// TwinCAT 3 PLC project controller
// ProgramVersion: 3.1.4024.0
// libraries:
//   mobject-collections, * (mobject)
//   mobject-commands, * (mobject)
//   mobject-disposable, * (mobject)
//   mobject-enumerable, * (mobject)
//   Tc2_ModbusSrv, * (Beckhoff Automation GmbH)
//   Tc3_Module, * (Beckhoff Automation GmbH)
//   Tc3_System, * (Beckhoff Automation GmbH)
// project tree:
//   Lib/ModbusTwin/ BasicModbusDigitalTwin.TcPOU
//   Lib/Modbus/ ModbusCommand.TcPOU, ReadRegistersCommand.TcPOU, WriteSingleRegisterCommand.TcPOU
//   Programs/ Main.TcPOU
//   Programs/TestTwin/ TestTwin.TcPOU, TestSlaveConfigData.TcDUT, TestSlaveFastDataA.TcDUT, TestSlaveFastDataB.TcDUT
//   _Tasks/ PlcTask.TcTTO (not stored)
// real-time tasks:
//   TASK PlcTask: cycle T#10ms, priority 20, ADS port 350

// ---- Programs/TestTwin/TestSlaveConfigData.TcDUT
TYPE TestSlaveConfigData :
STRUCT
	config1 : INT;
	config2 : INT;
END_STRUCT
END_TYPE

// ---- Programs/TestTwin/TestSlaveFastDataA.TcDUT
TYPE TestSlaveFastDataA :
STRUCT
	fastData1 : INT;
	fastData2 : INT;
END_STRUCT
END_TYPE

// ---- Programs/TestTwin/TestSlaveFastDataB.TcDUT
TYPE TestSlaveFastDataB :
STRUCT
	fastData3 : INT;
	fastData4 : INT;
END_STRUCT
END_TYPE

// ---- Lib/ModbusTwin/BasicModbusDigitalTwin.TcPOU
{attribute 'linkalways'} 
{attribute 'no_explicit_call' := 'This FB is a CLASS and must be accessed using methods or properties'}
{attribute 'enable_dynamic_creation'}
FUNCTION_BLOCK ABSTRACT BasicModbusDigitalTwin
VAR
	ipAddress : STRING(15);
	tcpPort : UINT := MODBUS_TCP_PORT;
	unitId : USINT;	

	cyclicCommands : LinkedList;
	queuedCommands : Queue;
	
	commandRunner : SingleAsyncCommandRunner;
	currentCommand : I_AsyncCommand;
END_VAR

METHOD PRIVATE AddCyclicalCommand
VAR_INPUT
	command : I_AsyncCommand;
END_VAR
cyclicCommands.AddItem(command);
END_METHOD

METHOD PROTECTED AddCyclicalReadRegisters
VAR_INPUT
	modbusAddress : UINT;
	quantity : UINT (1..128);	
	destinationAddress : POINTER TO BYTE;
	destinationLength : UDINT;
	timeout : TIME;
END_VAR
VAR
	_modbusAddress : UINT;
	_quantity : UINT (1..128);	
	_destinationAddress : POINTER TO BYTE;
	_destinationLength : UDINT;
	_timeout : TIME;
	pCommand : POINTER TO ReadRegistersCommand;
	command : I_AsyncCommand;
END_VAR
_modbusAddress := modbusAddress;
_quantity := quantity;
_destinationAddress := destinationAddress;
_destinationLength := destinationLength;
_timeout := timeout;

pCommand := __NEW(ReadRegistersCommand(
	ipAddress := THIS^.ipAddress, tcpPort := THIS^.tcpPort, unitId := THIS^.unitId,
	modbusAddress := _modbusAddress, quantity := _quantity,
	destinationAddress := _destinationAddress, destinationLength := _destinationLength,
	timeout := _timeout));
command := pCommand^;
AddCyclicalCommand(command);
END_METHOD

METHOD PUBLIC CyclicCall
VAR_INST
	cyclicEnumerator : I_ForwardEnumerator;

END_VAR
IF cyclicEnumerator = 0 THEN
	cyclicEnumerator := cyclicCommands.GetEnumerator();
END_IF

IF NOT commandRunner.Busy THEN
	IF queuedCommands.Count > 0 THEN
		IF queuedCommands.TryDequeue(currentCommand) THEN
			commandRunner.ExecuteCommand(currentCommand);
		END_IF		
	ELSE
		IF cyclicEnumerator.MoveNext() AND_THEN cyclicEnumerator.TryGet(currentCommand) THEN
			commandRunner.ExecuteCommand(currentCommand);
		ELSE
			cyclicEnumerator.Dispose();
			cyclicEnumerator := 0;
		END_IF
	END_IF
END_IF

commandRunner.CyclicCall();
END_METHOD

METHOD FB_init : BOOL
VAR_INPUT
	bInitRetains : BOOL; // if TRUE, the retain variables are initialized (warm start / cold start)
	bInCopyCode : BOOL;  // if TRUE, the instance afterwards gets moved into the copy code (online change)
	ipAddress : STRING(15);
	tcpPort : UINT := MODBUS_TCP_PORT;
	unitId : USINT;
END_VAR
THIS^.ipAddress := ipAddress;
THIS^.tcpPort := tcpPort;
THIS^.unitId := unitId;
END_METHOD

METHOD PRIVATE QueueCommand
VAR_INPUT
	command : I_AsyncCommand;
END_VAR
queuedCommands.Enqueue(command);
END_METHOD

METHOD PROTECTED QueueWriteSingleCoil
VAR_INPUT
	modbusAddress : WORD;
	value : BOOL;
	timeout : TIME;
END_VAR
VAR
	pCommand : POINTER TO WriteSingleRegisterCommand;
	command : I_AsyncCommand;
END_VAR
END_METHOD

METHOD PROTECTED QueueWriteSingleRegister
VAR_INPUT
	modbusAddress : UINT;
	data : WORD;
	timeout : TIME;
END_VAR
VAR
	_modbusAddress : UINT;
	_data : WORD;
	_timeout : TIME;
	pCommand : POINTER TO WriteSingleRegisterCommand;
	command : I_AsyncCommand;
END_VAR
_modbusAddress := modbusAddress;
_data := data;
_timeout := timeout;

pCommand := __NEW(WriteSingleRegisterCommand(
	ipAddress := THIS^.ipAddress, tcpPort := THIS^.tcpPort, unitId := THIS^.unitId,
	modbusAddress := _modbusAddress, data := _data,
	timeout := _timeout));
command := pCommand^;
QueueCommand(command);
END_METHOD

END_FUNCTION_BLOCK

// ---- Lib/Modbus/ReadRegistersCommand.TcPOU
{attribute 'linkalways'} 
{attribute 'no_explicit_call' := 'This FB is a CLASS and must be accessed using methods or properties'}
{attribute 'enable_dynamic_creation'}
FUNCTION_BLOCK ReadRegistersCommand EXTENDS ModbusCommand
VAR
	fb : FB_MBReadRegs;
END_VAR

METHOD FB_init : BOOL
VAR_INPUT
	bInitRetains : BOOL; // if TRUE, the retain variables are initialized (warm start / cold start)
	bInCopyCode : BOOL;  // if TRUE, the instance afterwards gets moved into the copy code (online change)
	ipAddress : STRING(15);
	tcpPort : UINT := MODBUS_TCP_PORT;
	unitId : USINT;
	modbusAddress : UINT;
	quantity : UINT (1..128);
	destinationAddress : POINTER TO BYTE;
	destinationLength : UDINT;
	timeout : TIME;
END_VAR
fb.sIPAddr := ipAddress;
fb.nTCPPort := tcpPort;
fb.nUnitID := USINT_TO_BYTE(unitId);
fb.nMBAddr := UINT_TO_WORD(modbusAddress);
fb.nQuantity := UINT_TO_WORD(quantity);
fb.pDestAddr := destinationAddress;
fb.cbLength := destinationLength;
fb.tTimeout := timeout;
END_METHOD

METHOD PROTECTED OnAborting
VAR_INPUT
	StateControl : I_AsyncCommandStateControl;
END_VAR
fb(bExecute := FALSE);
StateControl.Next();
END_METHOD

METHOD PROTECTED OnCompleting
VAR_INPUT
	StateControl : I_AsyncCommandStateControl;
END_VAR
fb(bExecute := FALSE);
StateControl.Next();
END_METHOD

METHOD PROTECTED OnErrored
fb(bExecute := FALSE);
END_METHOD

METHOD PROTECTED OnExecuting
VAR_INPUT
	StateControl : I_AsyncCommandStateControl;
END_VAR
fb(bExecute := TRUE);

IF NOT fb.bBusy THEN
	IF fb.bError THEN
		StateControl.Error(fb.nErrId);
	ELSE
		StateControl.Next();
	END_IF
END_IF
END_METHOD

METHOD PROTECTED OnIdle
fb(bExecute := FALSE);
END_METHOD

METHOD PROTECTED OnInitializing
VAR_INPUT
	StateControl : I_AsyncCommandStateControl;
END_VAR
fb(bExecute := TRUE);
StateControl.Next();
END_METHOD

END_FUNCTION_BLOCK

// ---- Lib/Modbus/ModbusCommand.TcPOU
{attribute 'linkalways'} 
{attribute 'no_explicit_call' := 'This FB is a CLASS and must be accessed using methods or properties'}
{attribute 'enable_dynamic_creation'}
FUNCTION_BLOCK ABSTRACT ModbusCommand EXTENDS AsyncCommand IMPLEMENTS I_Disposable

METHOD Dispose
__DELETE(THIS);
END_METHOD

METHOD FB_exit : BOOL
VAR_INPUT
	bInCopyCode : BOOL; // if TRUE, the exit method is called for exiting an instance that is copied afterwards (online change).
END_VAR
// by default you would return if this is an in copy code, i.e. online change to this class
IF bInCopyCode THEN
	RETURN;
END_IF

// A word of warning. FB_exit does not NOT operate in the same way as a typical inherited method. If a child class does not implement FB_exit then it does not
// gain this one for itself. 
// The system will automatically call each FB_exit on each layer of inheritance one by one, starting with the child class and making it's way to the parent.
// Therefore code in here will only be triggered once the system reaches this layer of the object's deletion. The child class and all of it's variables
// will already have had FB_exit called by the time we reach this point!
END_METHOD

END_FUNCTION_BLOCK

// ---- Lib/Modbus/WriteSingleRegisterCommand.TcPOU
{attribute 'linkalways'} 
{attribute 'no_explicit_call' := 'This FB is a CLASS and must be accessed using methods or properties'}
{attribute 'enable_dynamic_creation'}
FUNCTION_BLOCK WriteSingleRegisterCommand EXTENDS ModbusCommand
VAR
	fb : FB_MBWriteSingleReg;
END_VAR

METHOD FB_init : BOOL
VAR_INPUT
	bInitRetains : BOOL; // if TRUE, the retain variables are initialized (warm start / cold start)
	bInCopyCode : BOOL;  // if TRUE, the instance afterwards gets moved into the copy code (online change)
	ipAddress : STRING(15);
	tcpPort : UINT := MODBUS_TCP_PORT;
	unitId : USINT;
	modbusAddress : UINT;
	data : WORD;
	timeout : TIME;
END_VAR
fb.sIPAddr := ipAddress;
fb.nTCPPort := tcpPort;
fb.nUnitID := USINT_TO_BYTE(unitId);
fb.nMBAddr := UINT_TO_WORD(modbusAddress);
fb.nValue := data;
fb.tTimeout := timeout;
END_METHOD

METHOD PROTECTED OnAborting
VAR_INPUT
	StateControl : I_AsyncCommandStateControl;
END_VAR
fb(bExecute := FALSE);
StateControl.Next();
END_METHOD

METHOD PROTECTED OnCompleting
VAR_INPUT
	StateControl : I_AsyncCommandStateControl;
END_VAR
fb(bExecute := FALSE);
StateControl.Next();
END_METHOD

METHOD PROTECTED OnExecuting
VAR_INPUT
	StateControl : I_AsyncCommandStateControl;
END_VAR
fb(bExecute := TRUE);

IF NOT fb.bBusy THEN
	IF fb.bError THEN
		StateControl.Error(fb.nErrId);
	ELSE
		StateControl.Next();
	END_IF
END_IF
END_METHOD

METHOD PROTECTED OnIdle
fb(bExecute := FALSE);
END_METHOD

METHOD PROTECTED OnInitializing
VAR_INPUT
	StateControl : I_AsyncCommandStateControl;
END_VAR
fb(bExecute := TRUE);
StateControl.Next();
END_METHOD

END_FUNCTION_BLOCK

// ---- Programs/Main.TcPOU
PROGRAM Main
VAR
	testSlave : TestTwin(ipAddress := '127.0.0.1', tcpPort := 503, unitId := 255);
END_VAR

testSlave.CyclicCall();

END_PROGRAM

// ---- Programs/TestTwin/TestTwin.TcPOU
{attribute 'linkalways'} 
{attribute 'no_explicit_call' := 'This FB is a CLASS and must be accessed using methods or properties'}
{attribute 'enable_dynamic_creation'}
FUNCTION_BLOCK TestTwin EXTENDS BasicModbusDigitalTwin
VAR
	configData : TestSlaveConfigData;
	fastDataA : TestSlaveFastDataA;
	fastDataB : TestSlaveFastDataB;
	
	timeout : TIME := T#200MS;
END_VAR

{attribute 'monitoring' := 'call'}
PROPERTY PUBLIC Config1 : INT
GET // PUBLIC
Config1 := configData.config1;
END_GET
SET // PUBLIC
QueueWriteSingleRegister(0, INT_TO_WORD(Config1), timeout);
END_SET
END_PROPERTY

{attribute 'monitoring' := 'call'}
PROPERTY PUBLIC Config2 : INT
GET // PUBLIC
Config2 := configData.config2;
END_GET
SET // PUBLIC
QueueWriteSingleRegister(1, INT_TO_WORD(Config2), timeout);
END_SET
END_PROPERTY

{attribute 'monitoring' := 'call'}
PROPERTY PUBLIC Data1 : INT
GET // PUBLIC
Data1 := fastDataA.fastData1;
END_GET
SET // PUBLIC
QueueWriteSingleRegister(2, INT_TO_WORD(Data1), timeout);
END_SET
END_PROPERTY

{attribute 'monitoring' := 'call'}
PROPERTY PUBLIC Data2 : INT
GET // PUBLIC
Data2 := fastDataA.fastData2;
END_GET
SET // PUBLIC
QueueWriteSingleRegister(3, INT_TO_WORD(Data2), timeout);
END_SET
END_PROPERTY

{attribute 'monitoring' := 'call'}
PROPERTY PUBLIC Data3 : INT
GET // PUBLIC
Data3 := fastDataB.fastData3;
END_GET
SET // PUBLIC
QueueWriteSingleRegister(4, INT_TO_WORD(Data3), timeout);
END_SET
END_PROPERTY

{attribute 'monitoring' := 'call'}
PROPERTY PUBLIC Data4 : INT
GET // PUBLIC
Data4 := fastDataB.fastData4;
END_GET
SET // PUBLIC
QueueWriteSingleRegister(5, INT_TO_WORD(Data4), timeout);
END_SET
END_PROPERTY

METHOD FB_init : BOOL
VAR_INPUT
	bInitRetains : BOOL; // if TRUE, the retain variables are initialized (warm start / cold start)
	bInCopyCode : BOOL;  // if TRUE, the instance afterwards gets moved into the copy code (online change)
	ipAddress : STRING(15);
	tcpPort : UINT := MODBUS_TCP_PORT;
	unitId : USINT;
END_VAR
AddCyclicalReadRegisters(0, 2, ADR(configData), SIZEOF(configData), timeout);
AddCyclicalReadRegisters(2, 2, ADR(fastDataA), SIZEOF(fastDataA), timeout);
AddCyclicalReadRegisters(4, 2, ADR(fastDataB), SIZEOF(fastDataB), timeout);
END_METHOD

END_FUNCTION_BLOCK
